(* IEC 61131-3 sources: F100R_S278_Temperville/MyController.device.xml.v3^/Plc Logic.plclogic.xml.v3^/Application.application.xml.v3^/11_GestaoEnergetica, 3 files *)

(* ---- A_PricipalGestao.prg.st ---- *)
PROGRAM A_PricipalGestao
VAR
END_VAR

B_Acumuladores();
C_GerenciadorDatas();

(* ---- B_Acumuladores.prg.st ---- *)
PROGRAM B_Acumuladores
VAR
	rInstAquecimento : REAL;
	rInstDesligado : REAL;
	rInstOcioso : REAL;
	rInstTrabalhando : REAL;
	rInstTestando : REAL;
END_VAR

//--------------------- INICIO LÓGICA AQUECENDO ---------------------------\\

IF uStatusAquecimento = 1 THEN
	rInstAquecimento := (rBufferAquecendoDiario + rBufferDesligadoDiario + rBufferOciosoDiario + rBufferTestandoDiario + rBufferTrabalhandoDiario + rConsumoEnergiaReal_kWh) - rConsumoInicialDiario;
	rBufferAquecendoDiario := rBufferAquecendoDiario + rInstAquecimento;
ELSE
	rInstAquecimento := 0;
END_IF

//------------------------ FIM LÓGICA AQUECENDO ---------------------------\\

//--------------------- INICIO LÓGICA DESLIGADO ---------------------------\\

IF xResistenciasLigadas = FALSE AND NOT xTesteResistencias AND NOT xTesteEntradaSaidas THEN
	rInstDesligado := (rBufferAquecendoDiario + rBufferDesligadoDiario + rBufferOciosoDiario + rBufferTestandoDiario + rBufferTrabalhandoDiario + rConsumoEnergiaReal_kWh) - rConsumoInicialDiario;
	rBufferDesligadoDiario := rBufferDesligadoDiario + rInstDesligado;
END_IF

//------------------------ FIM LÓGICA DESLIGADO ---------------------------\\

//--------------------- INICIO LÓGICA OCIOSO ---------------------------\\

IF xResistenciasLigadas = TRUE AND uStatusMesaForno = 0 AND uStatusMesaResfriador = 0 THEN
	rInstOcioso := (rBufferAquecendoDiario + rBufferDesligadoDiario + rBufferOciosoDiario + rBufferTestandoDiario + rBufferTrabalhandoDiario + rConsumoEnergiaReal_kWh) - rConsumoInicialDiario;
	rBufferOciosoDiario := rBufferOciosoDiario + rInstOcioso;
ELSE
	rInstOcioso := 0;
END_IF

//------------------------ FIM LÓGICA OCIOSO ---------------------------\\

//--------------------- INICIO LÓGICA TRABALHANDO ----------------------\\

IF xResistenciasLigadas = TRUE AND uStatusMesaForno = 1 OR xResistenciasLigadas = TRUE AND uStatusMesaResfriador = 1 THEN
	rInstTrabalhando := (rBufferAquecendoDiario + rBufferDesligadoDiario + rBufferOciosoDiario + rBufferTestandoDiario + rBufferTrabalhandoDiario + rConsumoEnergiaReal_kWh) - rConsumoInicialDiario;
	rBufferTrabalhandoDiario := rBufferTrabalhandoDiario + rInstTrabalhando;
ELSE
	rInstTrabalhando := 0;
END_IF

//------------------------ FIM LÓGICA TRABALHANDO ----------------------\\

//--------------------- INICIO LÓGICA TESTANDO ----------------------\\

IF xResistenciasLigadas = FALSE AND xTesteResistencias OR xResistenciasLigadas = FALSE AND xTesteEntradaSaidas OR xOperacaoManual THEN
	rInstTestando := (rBufferAquecendoDiario + rBufferDesligadoDiario + rBufferOciosoDiario + rBufferTestandoDiario + rBufferTrabalhandoDiario + rConsumoEnergiaReal_kWh) - rConsumoInicialDiario;
	rBufferTestandoDiario := rBufferTestandoDiario + rInstTestando;
ELSE
	rInstTestando := 0;
END_IF

//------------------------ FIM LÓGICA TESTANDO -----------------------\\

(* ---- C_GerenciadorDatas.prg.st ---- *)
PROGRAM C_GerenciadorDatas
VAR
END_VAR

IF uDiaRealTime <> uDiaReferencia THEN

	rAquecendoDiario := rBufferAquecendoDiario;
	rBufferAquecendoDiario := 0;

	rDesligadoDiario := rBufferDesligadoDiario;
	rBufferDesligadoDiario := 0;

	rOciosoDiario := rBufferOciosoDiario;
	rBufferOciosoDiario := 0;

	rTestandoDiario := rBufferTestandoDiario;
	rBufferTestandoDiario := 0;

	rTrabalhandoDiario := rBufferTrabalhandoDiario;
	rBufferTrabalhandoDiario := 0;

	rConsumoInicialDiario := rConsumoEnergiaReal_kWh;

	uDiaReferencia := uDiaRealTime;

END_IF

IF uMesRealTime <> uMesReferencia THEN
	rAquecendoMensal := rBufferAquecendoMensal;
	rBufferAquecendoMensal := 0;

	rDesligadoMensal := rBufferDesligadoMensal;
	rBufferDesligadoMensal := 0;

	rOciosoMensal := rBufferOciosoMensal;
	rBufferOciosoMensal := 0;

	rTestandoMensal := rBufferTestandoMensal;
	rBufferTestandoMensal := 0;

	rTrabalhandoMensal := rBufferTrabalhandoMensal;
	rBufferTrabalhandoMensal := 0;

	bZeraAcumulado := TRUE;
	bGravaBancoE3 := TRUE;

ELSE
	uMesReferencia := uMesRealTime;
END_IF
